TYPE ST_HmiAlarmList :
STRUCT
	asAlarmList				: ARRAY[1..Param_Alarms.c_nMaxNrOfListEntries] OF STRING; // Active alarm texts for HMI list.
	sHighestActiveAlarm		: STRING; // Highest severity active alarm text.
END_STRUCT
END_TYPE

(* stored: Version 1.1.0.1, ProductVersion 3.1.4026.13
   DUT ST_HmiAlarmList: Id {32c735e7-89d0-463c-ab00-690f03812f39} *)
